INTERFACE I_Axis

END_INTERFACE

(* stored: Version 1.1.0.1, ProductVersion 3.1.4024.12
   Itf I_Axis: Id {0aa9fe18-9b82-4dd1-a575-8312f33b257a} *)
